PROGRAM TempChillerCtrl
VAR
	ARrStnChillerValueTempSetpointFinal: ARRAY [1..iStnQty] OF REAL;
	
END_VAR


(*Stn 3 Chiller Value Ctrl*)
IF bAutoPreparationPb  THEN
	ARrStnChillerValueTempSetpointFinal[3] := ARrStnTempSV[3] + ARrStnChillerValueTempSetpoint[3];
	
	IF ARrStnTempSV[3] >= ARrStnChillerValueTempSetpointFinal[3] THEN
	ARbStnChillerValueOnOff[3] := TRUE;
	ELSE 
	ARbStnChillerValueOnOff[3] := FALSE;
	END_IF

END_IF


ARwDO[eY13005_STN03CHILLEDWATERSUPPLYAV3_3].0 := ARbStnChillerValueOnOff[3];


(*Stn 6 Chiller Value Ctrl*)
IF bAutoPreparationPb  THEN
	ARrStnChillerValueTempSetpointFinal[6] := ARrStnTempSV[6] + ARrStnChillerValueTempSetpoint[6];
	
	IF ARrStnTempSV[6] >= ARrStnChillerValueTempSetpointFinal[6] THEN
	ARbStnChillerValueOnOff[6] := TRUE;
	ELSE 
	ARbStnChillerValueOnOff[6] := FALSE;
	END_IF

END_IF


ARwDO[eY13010_STN06CHILLEDWATERSUPPLYAV6_2].0 := ARbStnChillerValueOnOff[6];

END_PROGRAM

(* stored: Version 1.1.0.1, ProductVersion 3.1.4024.12
   POU TempChillerCtrl: Id {46a1d1b1-8d81-4299-bd24-7a5c4e10f8b7}, SpecialFunc None *)
